ST100_Modify_e.proceedOperation_1: (*  *)
    IF xIN_NextStep AND (GetTick() - iStartProcessTimeMili) >= (iProcessTimeMili1) THEN
        iStartProcessTimeMili := GetTick();
        iOUT_Step             := ST100_Modify_e.proceedOperation_2;
		_bBewegung := FALSE;
		
    ELSIF __ISVALIDREF(Mover) THEN
        IF Mover.MoverAxis.isInPos THEN
            IF _bBewegung THEN
               // Mover.MoverAxis.RelMoveTo(_bBewegungDist);
            ELSE
                //Mover.MoverAxis.RelMoveTo(-_bBewegungDist);
            END_IF

            _bBewegung := NOT _bBewegung;
        END_IF;
    END_IF;

ST100_Modify_e.proceedOperation_2: (*  *)
    IF xIN_NextStep AND (GetTick() - iStartProcessTimeMili) >= (iProcessTimeMili2) THEN
        iOUT_Step := ST100_Modify_e.SYNC_MOVER_LEAVE;
    END_IF;

ST100_Modify_e.SYNC_MOVER_LEAVE:
    // The mover needs to be taken by MoverMan
    IF NOT __ISVALIDREF(Mover) THEN
        iOUT_Step := ST100_Unload_e.DONE;
    END_IF

(***** DONE *****)
ST100_Modify_e.DONE: (* Letzter Schritt  *)
    IF NOT xIN_AlarmAktiv THEN
        //AUTO
        IF (enIN_State = StateAUTO) AND xIN_RestartCYCL THEN
            iOUT_Step := ST100_Modify_e.START;
            //STEP / END / LEERFAHREN restart
        ELSIF (enIN_State < StateAUTO) AND (enIN_State >= enState.StateSTEP) AND xIN_RestartCYCL THEN
            iOUT_Step := ST100_Modify_e.START;
            //STEP / END / LEERFAHREN fertig
        ELSIF (enIN_State = StateREADY) THEN
            iOUT_Step := ST100_Modify_e.READY;
        END_IF;
    END_IF;

(************ ERROR *************)
ST100_Modify_e.ERROR: (* ERROR *) ;

END_CASE;

END_FUNCTION_BLOCK

// ---- POUs/20_AUTO/FileMan/FB_FileMan.TcPOU
FUNCTION_BLOCK FB_FileMan
VAR_INPUT
    sPathName   : STRING; //
    bSave       : BOOL;
    bLoad       : BOOL;
    sRefString  : POINTER TO STRING(2000);
    uiStringLen : DINT; // string length
END_VAR
VAR_OUTPUT
    bError   : BOOL;  // true when a FB is in error (all fb are mixed here)
    nErrorId : UDINT; // the error id from the fb in error (all fb are mixed here)

    currentState : INT; // current state of this FB, use it for debug
END_VAR
VAR
    fb_open  : FB_FileOpen;
    fb_write : FB_FileWrite;
    fb_read  : FB_FileRead;
    fb_close : FB_FileClose;
    hFile    : UINT; // file number holder for write operation
    state    : INT := 0;

    bOpState : INT;   //0 = saving operation, 1 = loading operation, other = error
    nMode    : DWORD; // file open monde, depending on the command

    byteRead : UDINT; //number of byte read so far
END_VAR


CASE state OF

0: (* wait for operation *)
    IF bSave THEN
        state    := 1;
        bOpState := 0;
        nMode    := FOPEN_MODEWRITE;
    ELSIF bLoad THEN
        state    := 1;
        bOpState := 1;
        nMode    := FOPEN_MODEREAD;
    END_IF

1: (* open *)
    fb_open(sNetId    := '',
            sPathName := sPathName,
            nMode     := nMode,
            ePath     := PATH_GENERIC,
            bExecute  := TRUE,
            tTimeout  := T#3S,
            bBusy     =>,
            bError    =>,
            nErrId    =>,
            hFile     => hFile);

    IF NOT fb_open.bBusy THEN
        fb_open(bExecute := FALSE);

        IF 0 = bOpState THEN
            state := 3;
        ELSIF 1 = bOpState THEN
            state    := 5;
            byteRead := 0;
        END_IF
    END_IF

3: (* write *)
    fb_write(sNetId     := '',
             hFile      := hFile,
             pWriteBuff := sRefString,
             cbWriteLen := TO_UDINT(uiStringLen),
             bExecute   := TRUE,
             tTimeout   := T#3S,
             bBusy      =>,
             bError     =>,
             nErrId     =>,
             cbWrite    =>);

    IF NOT fb_write.bBusy THEN
        fb_write(bExecute := FALSE);
        state := 10;
    END_IF

5: (* read 100 bytes *)
    IF fb_read.bEOF THEN
        state := 9;
    ELSE
        fb_read(sNetId    := '',
                hFile     := hFile,
                pReadBuff := sRefString,
                cbReadLen := TO_UDINT(uiStringLen),
                bExecute  := TRUE,
                tTimeout  :=,
                bBusy     =>,
                bError    =>,
                nErrId    =>,
                cbRead    => byteRead,
                bEOF      =>);

        state := 6;
    END_IF

6: (* open *)
    fb_read(bExecute := FALSE);
    state := 5;

9:
    state := 10;

10: (* open *)
    fb_close(sNetId   := '',
             hFile    := hFile,
             bExecute := TRUE,
             tTimeout := T#3S,
             bBusy    =>,
             bError   =>,
             nErrId   =>);

    IF NOT fb_close.bBusy AND NOT bSave AND NOT bLoad THEN
        fb_close(bExecute := FALSE);
        state := 0;
    END_IF

END_CASE

bError       := fb_open.bError OR fb_write.bError OR fb_read.bError OR fb_close.bError;
nErrorId     := fb_open.nErrId OR fb_write.nErrId OR fb_read.nErrId OR fb_close.nErrId;
currentState := state;

END_FUNCTION_BLOCK

// ---- POUs/20_AUTO/FileMan/FB_ReadJSON.TcPOU
{attribute 'c++_compatible'}
FUNCTION_BLOCK FB_ReadJSON IMPLEMENTS ITcJsonSaxHandler
VAR_INPUT
    myArrayInput1 : REFERENCE TO ARRAY[1..CONSt.STATION_NUMBER] OF DINT;
    myArrayInput2 : REFERENCE TO ARRAY[1..CONSt.STATION_NUMBER] OF DINT;
END_VAR
VAR_OUTPUT
END_VAR
VAR
    iArrayIndex : INT;
	iArrayNumber : INT := 0;
END_VAR

{attribute 'TcTypeSystem'}
{attribute 'no-analysis'}
{attribute 'c++_compatible'}
{attribute 'minimal_input_size' := '4'}
{attribute 'pack_mode' := '4'}
METHOD OnBool : HRESULT
VAR_INPUT
	value	: BOOL;
END_VAR
END_METHOD

{attribute 'TcTypeSystem'}
{attribute 'no-analysis'}
{attribute 'c++_compatible'}
{attribute 'minimal_input_size' := '4'}
{attribute 'pack_mode' := '4'}
METHOD OnDint : HRESULT
VAR_INPUT
	value	: DINT;
END_VAR
END_METHOD

{attribute 'TcTypeSystem'}
{attribute 'no-analysis'}
{attribute 'c++_compatible'}
{attribute 'minimal_input_size' := '4'}
{attribute 'pack_mode' := '4'}
METHOD OnEndArray : HRESULT
VAR_INPUT
	elementCount	: UDINT;
END_VAR
OnEndArray := S_OK;
END_METHOD

{attribute 'TcTypeSystem'}
{attribute 'no-analysis'}
{attribute 'c++_compatible'}
{attribute 'minimal_input_size' := '4'}
{attribute 'pack_mode' := '4'}
METHOD OnEndObject : HRESULT
VAR_INPUT
	memberCount	: UDINT;
END_VAR
OnEndObject := S_OK;
END_METHOD

{attribute 'TcTypeSystem'}
{attribute 'no-analysis'}
{attribute 'c++_compatible'}
{attribute 'minimal_input_size' := '4'}
{attribute 'pack_mode' := '4'}
METHOD OnKey : HRESULT
VAR_IN_OUT CONSTANT
	key	: STRING;
END_VAR
VAR_INPUT
	len	: UDINT;
END_VAR
OnKey := S_OK;
END_METHOD

{attribute 'TcTypeSystem'}
{attribute 'no-analysis'}
{attribute 'c++_compatible'}
{attribute 'minimal_input_size' := '4'}
{attribute 'pack_mode' := '4'}
METHOD OnLint : HRESULT
VAR_INPUT
	value	: LINT;
END_VAR
END_METHOD

{attribute 'TcTypeSystem'}
{attribute 'no-analysis'}
{attribute 'c++_compatible'}
{attribute 'minimal_input_size' := '4'}
{attribute 'pack_mode' := '4'}
METHOD OnLreal : HRESULT
VAR_INPUT
	value	: LREAL;
END_VAR
END_METHOD

{attribute 'TcTypeSystem'}
{attribute 'no-analysis'}
{attribute 'c++_compatible'}
{attribute 'minimal_input_size' := '4'}
{attribute 'pack_mode' := '4'}
METHOD OnNull : HRESULT
END_METHOD

{attribute 'TcTypeSystem'}
{attribute 'no-analysis'}
{attribute 'c++_compatible'}
{attribute 'minimal_input_size' := '4'}
{attribute 'pack_mode' := '4'}
METHOD OnRawNumber : HRESULT
VAR_IN_OUT CONSTANT
	value	: STRING;
END_VAR
VAR_INPUT
	len	: UDINT;
END_VAR
END_METHOD

{attribute 'TcTypeSystem'}
{attribute 'no-analysis'}
{attribute 'c++_compatible'}
{attribute 'minimal_input_size' := '4'}
{attribute 'pack_mode' := '4'}
METHOD OnStartArray : HRESULT
THIS^.iArrayIndex := 1;
THIS^.iArrayNumber := THIS^.iArrayNumber + 1;
OnStartArray := S_OK;
END_METHOD

{attribute 'TcTypeSystem'}
{attribute 'no-analysis'}
{attribute 'c++_compatible'}
{attribute 'minimal_input_size' := '4'}
{attribute 'pack_mode' := '4'}
METHOD OnStartObject : HRESULT
OnStartObject := S_OK;
END_METHOD

{attribute 'TcTypeSystem'}
{attribute 'no-analysis'}
{attribute 'c++_compatible'}
{attribute 'minimal_input_size' := '4'}
{attribute 'pack_mode' := '4'}
METHOD OnString : HRESULT
VAR_IN_OUT CONSTANT
	value	: STRING;
END_VAR
VAR_INPUT
	len	: UDINT;
END_VAR
END_METHOD

{attribute 'TcTypeSystem'}
{attribute 'no-analysis'}
{attribute 'c++_compatible'}
{attribute 'minimal_input_size' := '4'}
{attribute 'pack_mode' := '4'}
METHOD OnUdint : HRESULT
VAR_INPUT
	value	: UDINT;
END_VAR
IF THIS^.iArrayNumber = 1 THEN
    THIS^.myArrayInput1[THIS^.iArrayIndex] := TO_DINT(value);
    THIS^.iArrayIndex                      := THIS^.iArrayIndex + 1;
ELSIF THIS^.iArrayNumber = 2 THEN
    THIS^.myArrayInput2[THIS^.iArrayIndex] := TO_DINT(value);
    THIS^.iArrayIndex                      := THIS^.iArrayIndex + 1;
END_IF
OnUdint := S_OK;
END_METHOD

{attribute 'TcTypeSystem'}
{attribute 'no-analysis'}
{attribute 'c++_compatible'}
{attribute 'minimal_input_size' := '4'}
{attribute 'pack_mode' := '4'}
METHOD OnUlint : HRESULT
VAR_INPUT
	value	: ULINT;
END_VAR
END_METHOD

{attribute 'TcTypeSystem'}
{attribute 'no-analysis'}
{attribute 'c++_compatible'}
{attribute 'minimal_input_size' := '4'}
{attribute 'pack_mode' := '4'}
METHOD TcAddRef : UDINT
END_METHOD

{attribute 'TcTypeSystem'}
{attribute 'no-analysis'}
{attribute 'c++_compatible'}
{attribute 'minimal_input_size' := '4'}
{attribute 'pack_mode' := '4'}
METHOD TcQueryInterface : HRESULT
VAR_INPUT
	iid	: REFERENCE TO IID;
	pipItf	: POINTER TO PVOID;
END_VAR
END_METHOD

{attribute 'TcTypeSystem'}
{attribute 'no-analysis'}
{attribute 'c++_compatible'}
{attribute 'minimal_input_size' := '4'}
{attribute 'pack_mode' := '4'}
METHOD TcRelease : UDINT
END_METHOD

END_FUNCTION_BLOCK

// ---- POUs/20_AUTO/FileMan/LoadFromMemory.TcPOU
FUNCTION LoadFromMemory : BOOL
VAR_INPUT
    sData : REFERENCE TO STRING(2000);
END_VAR
VAR
    fbJson     : FB_JsonSaxReader;
    pJsonParse : FB_ReadJSON;

    i : int;
END_VAR

pJsonParse.myArrayInput1 REF= PERS.iStationTimeDef1;
pJsonParse.myArrayInput2 REF= PERS.iStationTimeDef2;
fbJson.Parse(sJson := sData, ipHdl := pJsonParse);

END_FUNCTION

// ---- POUs/20_AUTO/FileMan/SaveInMemory.TcPOU
FUNCTION SaveInMemory : BOOL
VAR_INPUT
    sData : REFERENCE TO STRING(2000);
END_VAR
VAR
    fbJson     : FB_JsonSaxWriter;
    i          : int;
END_VAR

fbJson.ResetDocument();
// global object
fbJson.StartObject();
fbJson.AddKey('StationTimeArray');

// array1
fbJson.StartObject();
fbJson.AddKey('StationTime1');
fbJson.StartArray();

FOR i := 1 TO CONST.STATION_NUMBER BY 1 DO
    fbJson.AddDint(PERS.iStationTimeDef1[i]);
END_FOR

fbJson.EndArray();

// array2
fbJson.AddKey('StationTime2');
fbJson.StartArray();

FOR i := 1 TO CONST.STATION_NUMBER BY 1 DO
    fbJson.AddDint(PERS.iStationTimeDef2[i]);
END_FOR

fbJson.EndArray();
fbJson.EndObject();

fbJson.EndObject();
// end global object

// end of file
sData := fbJson.GetDocument();

fbJson.ResetDocument();

END_FUNCTION

// ---- POUs/20_AUTO/Mover/FB_PieceHolder.TcPOU
FUNCTION_BLOCK FB_PieceHolder IMPLEMENTS IObject
VAR_INPUT
END_VAR
VAR_OUTPUT
END_VAR
VAR
	_lrPosOffset : LREAL; // current offset position
	
	_iID : INT := 0; // instance ID, is set during FB_Init using the value of _iInstanceCounter 
END_VAR
VAR_STAT
	_iInstanceCounter : INT := 1; // instance counter
END_VAR

METHOD Equals : BOOL
VAR_INPUT
    object : ANY;
END_VAR
Equals := THIS = object.pValue;
END_METHOD

METHOD FB_init : BOOL
VAR_INPUT
    bInitRetains : BOOL;  // if TRUE, the retain variables are initialized (warm start / cold start)
    bInCopyCode  : BOOL;  // if TRUE, the instance afterwards gets moved into the copy code (online change)
    offset       : LREAL; //position offset of the tool using this toolhead, a negative value represents a move on the left
END_VAR
THIS^._iID := THIS^._iInstanceCounter;
THIS^._iInstanceCounter := THIS^._iInstanceCounter +1;
THIS^.PosOffset := offset;
END_METHOD

PROPERTY PosOffset : LREAL
GET
PosOffset := _lrPosOffset;
END_GET
SET
_lrPosOffset := PosOffset;
END_SET
END_PROPERTY

METHOD ToString : STRING
VAR_INPUT
END_VAR
ToString := CONCAT('FB_PieceHolder_', TO_STRING(THIS^._iID));
END_METHOD

END_FUNCTION_BLOCK

// ---- POUs/20_AUTO/Mover/FB_SortMoverByPos.TcPOU
FUNCTION_BLOCK FB_SortMoverByPos EXTENDS FB_Sort
VAR_INPUT
END_VAR
VAR_OUTPUT
END_VAR
VAR
END_VAR

(* Please override this method so it returns:
* 0 : a == b
*-1 : a < b
* 1 : a > b
* which a and b are the ADDRESS of the 2 elements you want to compare
*)
METHOD Compare : DINT
VAR_INPUT
	a : PVOID;
	b : PVOID;
END_VAR
VAR
    MoverDict_a : MoverDict;
    MoverDict_b : MoverDict;
END_VAR
Tc2_System.MEMCPY(ADR(MoverDict_a), a, SIZEOF(MoverDict));
Tc2_System.MEMCPY(ADR(MoverDict_b), b, SIZEOF(MoverDict));

IF MoverDict_a.MoverPos < MoverDict_b.MoverPos THEN
    Compare := -1;

ELSIF MoverDict_a.MoverPos > MoverDict_b.MoverPos THEN
    Compare := 1;

ELSE
    Compare := 0;

END_IF
END_METHOD

END_FUNCTION_BLOCK

// ---- POUs/20_AUTO/ST100/FB_ABL_100.TcPOU
FUNCTION_BLOCK FB_ABL_100
(****************************************************************************************)
(*	TITEL				Bezeichnung Ablauf	    										*)
(*	Status				ungetestet                         								*)
(*  Version:			1.0																*)
(*	Beschrieb:			Ablaufbeschreibung												*)
(*																						*)
(*	Steps:																				*)
(*		RESET:=0		Reset der Station												*)
(* 		INIT:=100		Initialisieren													*)
(*		... 			...																*)
(*		READY:=999		Initialisiert, Bereit für Start									*)
(*		START:=1000		Start Zyklisch 													*)
(*		... 			...																*)
(*		DONE:=8000		Letzer Schritt													*)
(*		ERROR:=9000		ALARM/Fehler													*)
(* 	09.09.2019/Dj																		*)
(***********************************Revisionen*******************************************)
(*	dd.mm.yyyy   KZ    x.y			Beschrieb											*)
(****************************************************************************************)

VAR_INPUT
    xIN_Reset       : BOOL;          // Schrittkette zurücksetzen 
    xIN_Init        : BOOL;          // Initialisieren
    xIN_Quit        : BOOL;          // Fehler quittieren 
    xIN_Start       : BOOL;          // Startbefehl
    xIN_Sperre      : BOOL;          // FB Sperren 
    xIN_NextStep    : BOOL;          // Nächsten Schritt ausführen 
    xIN_AlarmAktiv  : BOOL;          // Anlage hat Alarm
    xIN_DryCycle    : BOOL;          // Fahren ohne Teile
    xIN_RestartCYCL : BOOL;          // Zyklus erneut starten im STEP, END, LEERFAHREN
    xIN_MoverInPos  : BOOL;          // Set this flag when a mover is in position and ready to be handled
    enIN_State      : enState;       // Status Anlage
    tIN_Timeout     : TIME := T#10s; // Timout

    pxFG_Freigabe : POINTER TO BOOL; //Freigabe von Station

    // Application specific
    iProcessTimeMili : UDINT := 5000; // user defined station duration, in milisecond
END_VAR
VAR_OUTPUT
    (* standart Ausgänge *)
    xOUT_ErrFlag   : BOOL;   // Error Flag 
    xOUT_Busy      : BOOL;   // Baustein befindet sich im Ablauf 
    xOUT_Done      : BOOL;   // Baustein hat den Ablauf beendet 		
    xOUT_Ready     : BOOL;   // Ready to begin, should be the same state as done	
    xOUT_Timeout   : BOOL;   // Timeout FB 
    xOUT_InitDone  : BOOL;   // initialisierung fertig
    xOUT_Wait      : BOOL;   // Wartet auf Bedingung
    xOUT_MoverFree : BOOL;   // The mover is free to move
    iOUT_Step      : INT;    // Aktueller Schritt 
    sOUT_Step      : STRING; // Aktueller Schritt but in string format
    bOUT_Error     : BYTE;   // Fehlernummer

    iOUT_ProcessCompletion : INT; //process completion, express in % (0-100)
END_VAR
VAR
    (* Standard *)
    (* Schritt *)
    iLastStep : INT; // Merker letzter Schritt 
    iPreStep  : INT; // Schritt zurück nach Alarm 
    iAktStep  : INT; // aktueller Schritt

    // Trigger Starten 
    rtSTART : R_TRIG;
    // Timer TimeOut 
    TON_Timeout : TON;

    (* Bausteine *)

    (* Spezial *)
    iStartProcessTimeMili : UDINT; // start of the processing time, accurate at 100ns 

END_VAR
VAR CONSTANT
END_VAR

(*******************************************************************)
(* Trigger  *)
(*******************************************************************)
(* Zurücksetzen *)
IF xIN_RESET THEN
    iPreStep  := ST100_e.RESET;
    iOUT_Step := ST100_e.RESET;
END_IF;

(* Error Quittieren *)
IF (bOUT_Error <> 0) AND xIN_Quit THEN
    xOUT_ErrFlag := FALSE;
    bOUT_Error   := 0;
    iOUT_Step    := iPreStep;
END_IF;

(*******************************************************************)
(* Timer *)
(*******************************************************************)
TON_Timeout(IN := xIN_NextStep AND (iLastStep = iOUT_Step) (*todo FG *) ,
            PT := tIN_Timeout);

(*******************************************************************)
(* Bausteine *)
(*******************************************************************)

(*******************************************************************)
(* OUTPUTS *)
(*******************************************************************)
// Error Flag 
xOUT_ErrFlag := (bOUT_Error <> 0);
// Baustein befindet sich im Ablauf 
xOUT_Busy := (iOUT_Step > ST100_e.READY) AND (iOUT_Step < ST100_e.DONE);
// Baustein hat den Ablauf beendet
xOUT_Done := (iOUT_Step = ST100_e.DONE);
// Process ready
xOUT_Ready := (iOUT_Step = ST100_e.READY);
// Timeout FB 				 		
xOUT_Timeout := TON_Timeout.Q;
// Itialisierung fertig			
xOUT_InitDone := (iOUT_Step = ST100_e.READY);
// Aktueller Schritt			
iOUT_Step := iOUT_Step; //Im Ablauf gesetzt		
sOUT_Step := TO_STRING(iOUT_Step);
//Fehlernummer	 
bOUT_Error := bOUT_Error; //Im Ablauf/FB gesetzt	
(* Warte (alle Schritte wo auf FG oder Teile gewartet wird) *)
xOUT_Wait := (iOUT_Step = ST100_e.DONE);

xOUT_MoverFree := iOUT_Step >= ST100_e.MOVER_FREE_OP AND iOUT_Step < ST100_e.MOVER_NEEDED_OP;

IF iAktStep < ST100_e.START THEN
    iOUT_ProcessCompletion := 0;
ELSIF iAktStep > ST100_e.DONE THEN
    iOUT_ProcessCompletion := getPercent(iPreStep, TO_INT(ST100_e.START), TO_INT(ST100_e.proceedOperation_2) + 1);
ELSIF ST100_e.DONE = iAktStep THEN
    iOUT_ProcessCompletion := 100;
ELSE
    // iOUT_ProcessCompletion := getPercent(iAktStep, TO_INT(ST100_e.START), TO_INT(ST100_e.releaseMover) + 1);
    IF iProcessTimeMili > 0 THEN
        IF iAktStep < ST100_e.proceedOperation_1 THEN
            iOUT_ProcessCompletion := 0;
        ELSIF iAktStep = ST100_e.proceedOperation_1 THEN
            iOUT_ProcessCompletion := TO_INT(((GetTick() - iStartProcessTimeMili) * 100) / iProcessTimeMili);
        ELSIF iAktStep = ST100_e.proceedOperation_2 THEN
            iOUT_ProcessCompletion := 50 + TO_INT(((GetTick() - iStartProcessTimeMili) * 100) / iProcessTimeMili);
        ELSE
            iOUT_ProcessCompletion := 50;
        END_IF
    ELSE
        iOUT_ProcessCompletion := 0;
    END_IF
END_IF

(*******************************************************************)
(* Ablauf *)
(*******************************************************************)

(* Sperren *)
IF xIN_Sperre THEN
    iPreStep  := ST100_e.RESET;
    iOUT_Step := ST100_e.RESET;
    RETURN;
END_IF;

(* Schritt Merker *)
IF iAktStep <> iOUT_Step THEN
    iLastStep := iAktStep;
    iAktStep  := iOUT_Step;
END_IF

(* START *)
rtSTART(CLK := xIN_Start);

(*******************************************************************)
(* Schrittkette  *)
(*******************************************************************)
CASE iOUT_Step OF

(***** RESET *****)
ST100_e.RESET: (* Schritt 0-99 *)
    //Initialisierungen
    //Start Init Ablauf
    IF xIN_Init THEN
        iOUT_Step := ST100_e.INIT;
        //Start Manu Ablauf
    ELSIF enIN_State = StateMANU AND xIN_NextStep THEN
        iOUT_Step := ST100_e.INIT;
    END_IF;

(***** INIT *****)
ST100_e.INIT: (* Grundstellung ? *)
    IF TRUE THEN
        iOUT_Step := ST100_e.READY;
    ELSE
        iOUT_Step := ST100_e.INIT;
    END_IF;

(***** READY / INIT DONE *****)
ST100_e.READY:        (* Start AUTO,END,LEER,STEP *)
    IF xIN_Start THEN //IF rtSTART.Q THEN
        iOUT_Step := ST100_e.START;
    END_IF

(***** START  ZYKLISCH *****)
ST100_e.START: (*  *)
    IF xIN_NextStep AND pxFG_Freigabe^ THEN
        iOUT_Step             := ST100_e.proceedOperation_1;
        iStartProcessTimeMili := GetTick();
    END_IF;

ST100_e.proceedOperation_1: (*  *)
    IF xIN_NextStep AND (GetTick() - iStartProcessTimeMili) >= (iProcessTimeMili / 2) THEN
        iOUT_Step := ST100_e.waitOnMover;
    END_IF;

ST100_e.waitOnMover: (*  *)
    IF xIN_NextStep AND xIN_MoverInPos THEN
        iStartProcessTimeMili := GetTick();
        iOUT_Step             := ST100_e.proceedOperation_2;
    END_IF;

ST100_e.proceedOperation_2: (*  *)
    IF xIN_NextStep AND (GetTick() - iStartProcessTimeMili) >= (iProcessTimeMili / 2) THEN
        iOUT_Step := ST100_e.DONE;
    END_IF;

(***** DONE *****)
ST100_e.DONE: (* Letzter Schritt  *)
    IF NOT xIN_AlarmAktiv THEN
        //AUTO
        IF (enIN_State = StateAUTO) AND xIN_RestartCYCL THEN
            iOUT_Step := ST100_e.START;
            //STEP / END / LEERFAHREN restart
        ELSIF (enIN_State < StateAUTO) AND (enIN_State >= enState.StateSTEP) AND xIN_RestartCYCL THEN
            iOUT_Step := ST100_e.START;
            //STEP / END / LEERFAHREN fertig
        ELSIF (enIN_State = StateREADY) THEN
            iOUT_Step := ST100_e.READY;
        END_IF;
    END_IF;

(************ ERROR *************)
ST100_e.ERROR: (* ERROR *) ;

END_CASE;

END_FUNCTION_BLOCK

// ---- POUs/20_AUTO/TOOL/EqualApproximately.TcPOU
(*approximatelyEqual gives whether the difference between a and b is smaller than the acceptable
 error (epsilon), determined by the larger of a or b. This means that the two values are 
"close enough", and we can say that they're approximately equal.*)
FUNCTION EqualApproximately
VAR_INPUT
    a       : LREAL;
    b       : LREAL;
    epsilon : LREAL;
END_VAR
VAR
END_VAR

IF ABS(a) < ABS(b) THEN
    EqualApproximately := ABS(a - b) <= (ABS(b) * epsilon);
ELSE
    EqualApproximately := ABS(a - b) <= (ABS(a) * epsilon);
END_IF

END_FUNCTION

// ---- POUs/20_AUTO/TOOL/EqualEssentially.TcPOU
(*essentiallyEqual gives whether the difference between a and b is smaller than the acceptable error (epsilon), 
determined by the smaller of a or b. This means that the values differ less than the acceptable difference in 
any calculation, so that perhaps they're not actually equal, but they're "essentially equal" (given the epsilon). *)
FUNCTION EqualEssentially : BOOL
VAR_INPUT
    a       : LREAL;
    b       : LREAL;
    epsilon : LREAL;
END_VAR
VAR
END_VAR

IF ABS(a) > ABS(b) THEN
    EqualEssentially := ABS(a - b) <= (ABS(b) * epsilon);
ELSE
    EqualEssentially := ABS(a - b) <= (ABS(a) * epsilon);
END_IF

END_FUNCTION

// ---- GlobalTextList.TcGTLO
TEXTLIST GlobalTextList
  373 = '%d'
  962 = '%f'
  999 = '%s'
  454 = '4'
  166 = 'Acceleration:'
  629 = 'AUTO'
  404 = 'Avg'
  101 = 'Current state'
  998 = 'Current state:'
  203 = 'END'
  557 = 'INIT'
  820 = 'LEER'
  905 = 'MANU'
  641 = 'Max'
  23 = 'Max speed:'
  386 = 'Min'
  590 = 'Mover 1 actual pos'
  716 = 'Mover 1 actual pos :'
  357 = 'Mover n°'
  310 = 'Mover n°%d'
  821 = 'Mover n°%s'
  679 = 'Navette 1 Pos'
  378 = 'PERS.iStationTimeDef[1]'
  375 = 'Piece holder:'
  639 = 'Process name:'
  964 = 'Process time :'
  566 = 'QUIT'
  849 = 'RESET TEMP COUNTER'
  832 = 'Save var'
  105 = 'SET'
  630 = 'Set all mover ApproachScenario'
  84 = 'Set all station time'
  137 = 'ST100'
  367 = 'ST105'
  965 = 'ST110'
  902 = 'ST115'
  633 = 'ST120'
  304 = 'ST125'
  610 = 'ST130'
  108 = 'ST135'
  328 = 'ST140'
  559 = 'ST145'
  406 = 'ST150'
  30 = 'ST155'
  326 = 'ST160'
  841 = 'ST165'
  619 = 'ST170'
  492 = 'ST175'
  422 = 'ST176'
  415 = 'ST180'
  710 = 'ST185'
  151 = 'ST190'
  960 = 'ST200'
  20 = 'ST210'
  526 = 'ST220'
  583 = 'ST230'
  75 = 'ST240'
  706 = 'ST250'
  364 = 'ST260'
  34 = 'ST270'
  69 = 'ST290'
  840 = 'ST300'
  729 = 'ST60'
  992 = 'ST70'
  939 = 'START'
  702 = 'Station name:'
  645 = 'STEP'
  457 = 'STOP'
  58 = 'Stop mover'
  242 = '[ms]'
END_TEXTLIST

// ---- VISUs/VISU_main.TcVIS
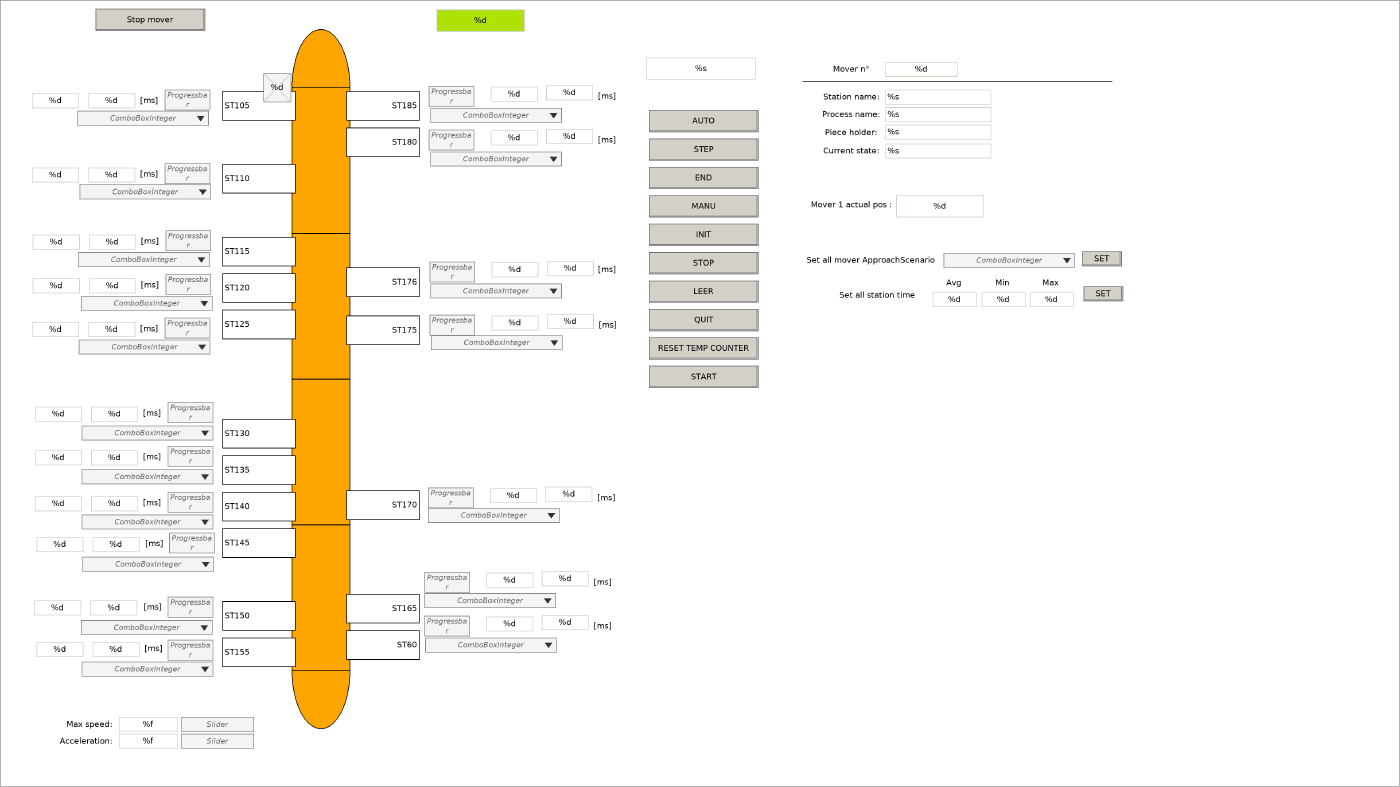
VISUALIZATION VISU_main  // 1920x1080
    Ellipse (400,840 80x160)
    Rectangle (400,720 80x200)
    Rectangle (400,520 80x200)
    Rectangle (400,320 80x200)
    Ellipse (400,40 80x160)
    Rectangle (400,120 80x200)
    Button (890,151 150x30), "AUTO", colour toggle: HMI.btArMain[0].on, input disabled if: HMI.btArMain[0].disable
        tap HMI.btArMain[0].button
    Button (890,190 150x30), "STEP", colour toggle: HMI.btArMain[1].on, input disabled if: HMI.btArMain[1].disable
        tap HMI.btArMain[1].button
    Button (890,229 150x30), "END", colour toggle: HMI.btArMain[2].on, input disabled if: HMI.btArMain[2].disable
        tap HMI.btArMain[2].button
    Button (890,307 150x30), "INIT", colour toggle: HMI.btArMain[4].on, input disabled if: HMI.btArMain[4].disable
        tap HMI.btArMain[4].button
    Button (890,346 150x30), "STOP", colour toggle: HMI.btArMain[5].disable, input disabled if: HMI.btArMain[5].disable
        tap HMI.btArMain[5].button
    Button (890,385 150x30), "LEER", colour toggle: HMI.btArMain[6].disable, input disabled if: HMI.btArMain[6].disable
        tap HMI.btArMain[6].button
    Button (890,424 150x30), "QUIT", colour toggle: HMI.btArMain[7].disable, input disabled if: HMI.btArMain[7].disable
        tap HMI.btArMain[7].button
    Button (890,463 150x30), "RESET TEMP COUNTER", colour toggle: HMI.btArMain[8].disable, input disabled if: HMI.btArMain[8].disable
        tap HMI.btArMain[8].button
    Button (890,268 150x30), "MANU", colour toggle: HMI.btArMain[3].on, input disabled if: HMI.btArMain[3].disable
        tap HMI.btArMain[3].button
    Textfield (886,79 150x30), "%s", text variable: _14_STATE.sStateDbg
    Button (890,502 150x30), "START", colour toggle: HMI.btArMain[9].disable, input disabled if: HMI.btArMain[9].disable
        tap HMI.btArMain[9].button
    Rectangle (475,175 100x40), "ST180", colour toggle: NOT PRG.st180_aut.xMoverPathFree
    Rectangle (475,367 100x40), "ST176", colour toggle: NOT PRG.st176_aut.xMoverPathFree
    Rectangle (475,433 100x40), "ST175", colour toggle: NOT PRG.st170_aut.xMoverPathFree
    Rectangle (475,673 100x40), "ST170", colour toggle: NOT PRG.st170_aut.xMoverPathFree
    Rectangle (475,815 100x40), "ST165", colour toggle: NOT PRG.st165_aut.xMoverPathFree
    Rectangle (475,865 100x40), "ST60", colour toggle: NOT PRG.st160_aut.xMoverPathFree
    Rectangle (305,875 100x40), "ST155", colour toggle: NOT PRG.st155_aut.xMoverPathFree
    Rectangle (475,125 100x40), "ST185", colour toggle: NOT PRG.st185_aut.xMoverPathFree
    Progressbar (588,178 62x28), variable: SIMU.iCompletionHMI[17]
    Progressbar (589,359 62x28), variable: SIMU.iCompletionHMI[16]
    Progressbar (589,432 62x28), variable: SIMU.iCompletionHMI[15]
    Progressbar (587,669 62x28), variable: SIMU.iCompletionHMI[14]
    Progressbar (582,785 62x28), variable: SIMU.iCompletionHMI[13]
    Progressbar (582,845 62x28), variable: SIMU.iCompletionHMI[12]
    Progressbar (230,878 62x28), variable: SIMU.iCompletionHMI[11]
    Progressbar (588,118 62x28), variable: SIMU.iCompletionHMI[18]
    Textfield (749,177 64x20), "%d", text variable: PERS.iStationTimeDef2[17]
        OnMouseDown: write the text variable via Default
    Label (805,177 55x30), "[ms]"
    Textfield (750,358 64x20), "%d", text variable: PERS.iStationTimeDef2[16]
        OnMouseDown: write the text variable via Default
    Label (805,355 55x30), "[ms]"
    Textfield (750,431 64x20), "%d", text variable: PERS.iStationTimeDef2[15]
        OnMouseDown: write the text variable via Default
    Label (806,431 55x30), "[ms]"
    Textfield (748,668 64x20), "%d", text variable: PERS.iStationTimeDef2[14]
        OnMouseDown: write the text variable via Default
    Label (804,668 55x30), "[ms]"
    Textfield (743,784 64x20), "%d", text variable: PERS.iStationTimeDef2[13]
        OnMouseDown: write the text variable via Default
    Label (799,784 55x30), "[ms]"
    Textfield (743,844 64x20), "%d", text variable: PERS.iStationTimeDef2[12]
        OnMouseDown: write the text variable via Default
    Label (799,844 55x30), "[ms]"
    Textfield (127,881 64x20), "%d", text variable: PERS.iStationTimeDef2[11]
        OnMouseDown: write the text variable via Default
    Label (183,875 55x30), "[ms]"
    Textfield (749,117 64x20), "%d", text variable: PERS.iStationTimeDef2[18]
        OnMouseDown: write the text variable via Default
    Label (805,117 55x30), "[ms]"
    Textfield (1229,268 120x30), "%d", text variable: MAIN.MoverMan._MoverList[1]._MoverAxis._CurrentPos
        OnMouseDown: write the text variable via Default
    Label (1080,266 146x30), "Mover 1 actual pos :"
    Textfield (599,13 120x30), "%d", text variable: PERS.iRecipeCurrent
        OnMouseDown: write the text variable via Default
    ComboBoxInteger (590,148 180x20), variable: MAIN.MoverMan._StationList[18]._ApproachScenario
    ComboBoxInteger (590,208 180x20), variable: MAIN.MoverMan._StationList[17]._ApproachScenario
    ComboBoxInteger (590,389 180x20), variable: MAIN.MoverMan._StationList[16]._ApproachScenario
    ComboBoxInteger (591,460 180x20), variable: MAIN.MoverMan._StationList[15]._ApproachScenario
    ComboBoxInteger (587,697 180x20), variable: MAIN.MoverMan._StationList[14]._ApproachScenario
    ComboBoxInteger (582,814 180x20), variable: MAIN.MoverMan._StationList[13]._ApproachScenario
    ComboBoxInteger (583,875 180x20), variable: MAIN.MoverMan._StationList[12]._ApproachScenario
    ComboBoxInteger (112,908 180x20), variable: MAIN.MoverMan._StationList[11]._ApproachScenario
    Rectangle (305,825 100x40), "ST150", colour toggle: NOT PRG.st150_aut.xMoverPathFree
    Progressbar (230,819 62x28), variable: SIMU.iCompletionHMI[10]
    Textfield (124,824 64x20), "%d", text variable: PERS.iStationTimeDef2[10]
        OnMouseDown: write the text variable via Default
    Label (182,818 55x30), "[ms]"
    ComboBoxInteger (111,851 180x20), variable: MAIN.MoverMan._StationList[10]._ApproachScenario
    Textfield (127,737 64x20), "%d", text variable: PERS.iStationTimeDef2[9]
        OnMouseDown: write the text variable via Default
    Label (184,731 55x30), "[ms]"
    Rectangle (305,725 100x40), "ST145", colour toggle: NOT PRG.st105_aut.xMoverPathFree
    Progressbar (232,731 62x28), variable: SIMU.iCompletionHMI[9]
    ComboBoxInteger (113,764 180x20), variable: MAIN.MoverMan._StationList[9]._ApproachScenario
    Textfield (125,681 64x20), "%d", text variable: PERS.iStationTimeDef2[8]
        OnMouseDown: write the text variable via Default
    Label (181,675 55x30), "[ms]"
    Rectangle (305,675 100x40), "ST140", colour toggle: NOT PRG.st140_aut.xMoverPathFree
    Progressbar (230,675 62x28), variable: SIMU.iCompletionHMI[8]
    ComboBoxInteger (112,706 180x20), variable: MAIN.MoverMan._StationList[8]._ApproachScenario
    Textfield (125,618 64x20), "%d", text variable: PERS.iStationTimeDef2[7]
        OnMouseDown: write the text variable via Default
    Label (181,612 55x30), "[ms]"
    Rectangle (305,625 100x40), "ST135", colour toggle: NOT PRG.st135_aut.xMoverPathFree
    Progressbar (230,612 62x28), variable: SIMU.iCompletionHMI[7]
    ComboBoxInteger (112,644 180x20), variable: MAIN.MoverMan._StationList[7]._ApproachScenario
    Textfield (125,558 64x20), "%d", text variable: PERS.iStationTimeDef2[6]
        OnMouseDown: write the text variable via Default
    Label (181,552 55x30), "[ms]"
    Rectangle (305,575 100x40), "ST130", colour toggle: NOT PRG.st130_aut.xMoverPathFree
    Progressbar (230,552 62x28), variable: SIMU.iCompletionHMI[6]
    ComboBoxInteger (112,584 180x20), variable: MAIN.MoverMan._StationList[6]._ApproachScenario
    Textfield (121,442 64x20), "%d", text variable: PERS.iStationTimeDef2[5]
        OnMouseDown: write the text variable via Default
    Label (177,436 55x30), "[ms]"
    Rectangle (305,425 100x40), "ST125", colour toggle: NOT PRG.st125_aut.xMoverPathFree
    Progressbar (226,436 62x28), variable: SIMU.iCompletionHMI[5]
    ComboBoxInteger (108,466 180x20), variable: MAIN.MoverMan._StationList[5]._ApproachScenario
    Textfield (122,382 64x20), "%d", text variable: PERS.iStationTimeDef2[4]
        OnMouseDown: write the text variable via Default
    Label (178,376 55x30), "[ms]"
    Rectangle (305,375 100x40), "ST120", colour toggle: NOT PRG.st120_aut.xMoverPathFree
    Progressbar (227,376 62x28), variable: SIMU.iCompletionHMI[4]
    ComboBoxInteger (111,406 180x20), variable: MAIN.MoverMan._StationList[4]._ApproachScenario
    Textfield (122,322 64x20), "%d", text variable: PERS.iStationTimeDef2[3]
        OnMouseDown: write the text variable via Default
    Label (178,316 55x30), "[ms]"
    Rectangle (305,325 100x40), "ST115", colour toggle: NOT PRG.st115_aut.xMoverPathFree
    Progressbar (227,316 62x28), variable: SIMU.iCompletionHMI[3]
    ComboBoxInteger (107,346 180x20), variable: MAIN.MoverMan._StationList[3]._ApproachScenario
    Textfield (121,230 64x20), "%d", text variable: PERS.iStationTimeDef2[2]
        OnMouseDown: write the text variable via Default
    Label (177,224 55x30), "[ms]"
    Rectangle (305,225 100x40), "ST110", colour toggle: NOT PRG.st110_aut.xMoverPathFree
    Progressbar (226,224 62x28), variable: SIMU.iCompletionHMI[2]
    ComboBoxInteger (109,253 180x20), variable: MAIN.MoverMan._StationList[2]._ApproachScenario
    Rectangle (305,125 100x40), "ST105", colour toggle: NOT PRG.st105_aut.xMoverPathFree
    Progressbar (226,123 62x28), variable: SIMU.iCompletionHMI[1]
    Textfield (121,128 64x20), "%d", text variable: PERS.iStationTimeDef2[1]
        OnMouseDown: write the text variable via Edit
    Label (177,123 55x30), "[ms]"
    ComboBoxInteger (106,152 180x20), variable: MAIN.MoverMan._StationList[1]._ApproachScenario
    ComboBoxInteger (1294,347 180x20), variable: MAIN.MoverMan.HMI_Scenario
    Label (1098,342 187x30), "Set all mover ApproachScenario"
    Button (1484,345 54x20), "SET"
        OnMouseDown: execute { MAIN.MoverMan.SetAllScenario(); }
    Label (1132,390 126x30), "Set all station time"
    Textfield (1279,401 60x20), "%d", text variable: MAIN.MoverMan.HMI_TimeAvg
        OnMouseDown: write the text variable via Default
    Label (1280,377 56x22), "Avg"
    Textfield (1346,401 60x20), "%d", text variable: MAIN.MoverMan.HMI_TimeMin
        OnMouseDown: write the text variable via Default
    Label (1347,377 56x22), "Min"
    Textfield (1412,401 60x20), "%d", text variable: MAIN.MoverMan.HMI_TimeMax
        OnMouseDown: write the text variable via Default
    Label (1413,377 56x22), "Max"
    Button (1486,393 54x20), "SET"
        OnMouseDown: execute { MAIN.MoverMan.SetAllTimers(ADR(PERS.iStationTimeDef1), 0); MAIN.MoverMan.SetAllTimers(ADR(PERS.iStationTimeDef2), 500); }
    Button (131,12 150x30), "Stop mover", colour toggle: MAIN.MoverMan.HMI_xStopMover
        toggle MAIN.MoverMan.HMI_xStopMover
    Label (1118,80 99x30), "Mover n°"
    Line (1101,111) (1525,111)
    Label (1118,118 99x30), "Station name:"
    Label (1118,142 99x30), "Process name:"
    Label (1118,167 99x30), "Piece holder:"
    Label (1118,192 99x30), "Current state:"
    Textfield (1214,85 99x20), "%d", text variable: MAIN.MoverMan.HMI_iSelMover
        OnMouseDown: write the text variable via Default
    Textfield (1214,123 145x20), "%s", text variable: MAIN.MoverMan._MoverList[MAIN.MoverMan.HMI_iSelMover].Station.ToString()
    Textfield (1214,147 145x20), "%s", text variable: MAIN.MoverMan._MoverList[MAIN.MoverMan.HMI_iSelMover].Station.Process.ToString()
    Textfield (1214,171 145x20), "%s"
    Textfield (1214,197 145x20), "%s", text variable: TO_STRING(MAIN.MoverMan._MoverList[MAIN.MoverMan.HMI_iSelMover]._State)
    Image (361,100 38x40), "%d", text variable: MAIN.MoverMan._MoverList[1]._ID, colour toggle: MAIN.MoverMan._SimuMoverList[1]._xStuck, invisible if: MAIN.MoverMan._MoverList[1]._MoverAxis._iID>CONST.MOVER_NUMBER, image: Custom.MoverSimu_final
        p3560616238: MAIN.MoverMan._MoverList[1]._MoverAxis.outSimuCurrentPos.x
        p2738717112: MAIN.MoverMan._MoverList[1]._MoverAxis.outSimuCurrentPos.y
        p2858320360: -MAIN.MoverMan._MoverList[1]._MoverAxis.outSimuCurrentRot
    Image (361,100 38x40), "%d", text variable: MAIN.MoverMan._MoverList[2]._ID, colour toggle: MAIN.MoverMan._SimuMoverList[2]._xStuck, invisible if: MAIN.MoverMan._MoverList[2]._MoverAxis._iID>CONST.MOVER_NUMBER, image: Custom.MoverSimu_final
        p3560616238: MAIN.MoverMan._MoverList[2]._MoverAxis.outSimuCurrentPos.x
        p2738717112: MAIN.MoverMan._MoverList[2]._MoverAxis.outSimuCurrentPos.y
        p2858320360: -MAIN.MoverMan._MoverList[2]._MoverAxis.outSimuCurrentRot
    Image (361,100 38x40), "%d", text variable: MAIN.MoverMan._MoverList[3]._ID, colour toggle: MAIN.MoverMan._SimuMoverList[3]._xStuck, invisible if: MAIN.MoverMan._MoverList[3]._MoverAxis._iID>CONST.MOVER_NUMBER, image: Custom.MoverSimu_final
        p3560616238: MAIN.MoverMan._MoverList[3]._MoverAxis.outSimuCurrentPos.x
        p2738717112: MAIN.MoverMan._MoverList[3]._MoverAxis.outSimuCurrentPos.y
        p2858320360: -MAIN.MoverMan._MoverList[3]._MoverAxis.outSimuCurrentRot
    Image (361,100 38x40), "%d", text variable: MAIN.MoverMan._MoverList[4]._ID, colour toggle: MAIN.MoverMan._SimuMoverList[4]._xStuck, invisible if: MAIN.MoverMan._MoverList[4]._MoverAxis._iID>CONST.MOVER_NUMBER, image: Custom.MoverSimu_final
        p3560616238: MAIN.MoverMan._MoverList[4]._MoverAxis.outSimuCurrentPos.x
        p2738717112: MAIN.MoverMan._MoverList[4]._MoverAxis.outSimuCurrentPos.y
        p2858320360: -MAIN.MoverMan._MoverList[4]._MoverAxis.outSimuCurrentRot
    Image (361,100 38x40), "%d", text variable: MAIN.MoverMan._MoverList[5]._ID, colour toggle: MAIN.MoverMan._SimuMoverList[5]._xStuck, invisible if: MAIN.MoverMan._MoverList[5]._MoverAxis._iID>CONST.MOVER_NUMBER, image: Custom.MoverSimu_final
        p3560616238: MAIN.MoverMan._MoverList[5]._MoverAxis.outSimuCurrentPos.x
        p2738717112: MAIN.MoverMan._MoverList[5]._MoverAxis.outSimuCurrentPos.y
        p2858320360: -MAIN.MoverMan._MoverList[5]._MoverAxis.outSimuCurrentRot
    Image (361,100 38x40), "%d", text variable: MAIN.MoverMan._MoverList[6]._ID, colour toggle: MAIN.MoverMan._SimuMoverList[6]._xStuck, invisible if: MAIN.MoverMan._MoverList[6]._MoverAxis._iID>CONST.MOVER_NUMBER, image: Custom.MoverSimu_final
        p3560616238: MAIN.MoverMan._MoverList[6]._MoverAxis.outSimuCurrentPos.x
        p2738717112: MAIN.MoverMan._MoverList[6]._MoverAxis.outSimuCurrentPos.y
        p2858320360: -MAIN.MoverMan._MoverList[6]._MoverAxis.outSimuCurrentRot
    Image (361,100 38x40), "%d", text variable: MAIN.MoverMan._MoverList[7]._ID, colour toggle: MAIN.MoverMan._SimuMoverList[7]._xStuck, invisible if: MAIN.MoverMan._MoverList[7]._MoverAxis._iID>CONST.MOVER_NUMBER, image: Custom.MoverSimu_final
        p3560616238: MAIN.MoverMan._MoverList[7]._MoverAxis.outSimuCurrentPos.x
        p2738717112: MAIN.MoverMan._MoverList[7]._MoverAxis.outSimuCurrentPos.y
        p2858320360: -MAIN.MoverMan._MoverList[7]._MoverAxis.outSimuCurrentRot
    Image (361,100 38x40), "%d", text variable: MAIN.MoverMan._MoverList[8]._ID, colour toggle: MAIN.MoverMan._SimuMoverList[8]._xStuck, invisible if: MAIN.MoverMan._MoverList[8]._MoverAxis._iID>CONST.MOVER_NUMBER, image: Custom.MoverSimu_final
        p3560616238: MAIN.MoverMan._MoverList[8]._MoverAxis.outSimuCurrentPos.x
        p2738717112: MAIN.MoverMan._MoverList[8]._MoverAxis.outSimuCurrentPos.y
        p2858320360: -MAIN.MoverMan._MoverList[8]._MoverAxis.outSimuCurrentRot
    Image (361,100 38x40), "%d", text variable: MAIN.MoverMan._MoverList[9]._ID, colour toggle: MAIN.MoverMan._SimuMoverList[9]._xStuck, invisible if: MAIN.MoverMan._MoverList[9]._MoverAxis._iID>CONST.MOVER_NUMBER, image: Custom.MoverSimu_final
        p3560616238: MAIN.MoverMan._MoverList[9]._MoverAxis.outSimuCurrentPos.x
        p2738717112: MAIN.MoverMan._MoverList[9]._MoverAxis.outSimuCurrentPos.y
        p2858320360: -MAIN.MoverMan._MoverList[9]._MoverAxis.outSimuCurrentRot
    Image (361,100 38x40), "%d", text variable: MAIN.MoverMan._MoverList[10]._ID, colour toggle: MAIN.MoverMan._SimuMoverList[10]._xStuck, invisible if: MAIN.MoverMan._MoverList[10]._MoverAxis._iID>CONST.MOVER_NUMBER, image: Custom.MoverSimu_final
        p3560616238: MAIN.MoverMan._MoverList[10]._MoverAxis.outSimuCurrentPos.x
        p2738717112: MAIN.MoverMan._MoverList[10]._MoverAxis.outSimuCurrentPos.y
        p2858320360: -MAIN.MoverMan._MoverList[10]._MoverAxis.outSimuCurrentRot
    Image (361,100 38x40), "%d", text variable: MAIN.MoverMan._MoverList[11]._ID, colour toggle: MAIN.MoverMan._SimuMoverList[11]._xStuck, invisible if: MAIN.MoverMan._MoverList[11]._MoverAxis._iID>CONST.MOVER_NUMBER, image: Custom.MoverSimu_final
        p3560616238: MAIN.MoverMan._MoverList[11]._MoverAxis.outSimuCurrentPos.x
        p2738717112: MAIN.MoverMan._MoverList[11]._MoverAxis.outSimuCurrentPos.y
        p2858320360: -MAIN.MoverMan._MoverList[11]._MoverAxis.outSimuCurrentRot
    Image (361,100 38x40), "%d", text variable: MAIN.MoverMan._MoverList[12]._ID, colour toggle: MAIN.MoverMan._SimuMoverList[12]._xStuck, invisible if: MAIN.MoverMan._MoverList[12]._MoverAxis._iID>CONST.MOVER_NUMBER, image: Custom.MoverSimu_final
        p3560616238: MAIN.MoverMan._MoverList[12]._MoverAxis.outSimuCurrentPos.x
        p2738717112: MAIN.MoverMan._MoverList[12]._MoverAxis.outSimuCurrentPos.y
        p2858320360: -MAIN.MoverMan._MoverList[12]._MoverAxis.outSimuCurrentRot
    Image (361,100 38x40), "%d", text variable: MAIN.MoverMan._MoverList[13]._ID, colour toggle: MAIN.MoverMan._SimuMoverList[13]._xStuck, invisible if: MAIN.MoverMan._MoverList[13]._MoverAxis._iID>CONST.MOVER_NUMBER, image: Custom.MoverSimu_final
        p3560616238: MAIN.MoverMan._MoverList[13]._MoverAxis.outSimuCurrentPos.x
        p2738717112: MAIN.MoverMan._MoverList[13]._MoverAxis.outSimuCurrentPos.y
        p2858320360: -MAIN.MoverMan._MoverList[13]._MoverAxis.outSimuCurrentRot
    Image (361,100 38x40), "%d", text variable: MAIN.MoverMan._MoverList[14]._ID, colour toggle: MAIN.MoverMan._SimuMoverList[14]._xStuck, invisible if: MAIN.MoverMan._MoverList[14]._MoverAxis._iID>CONST.MOVER_NUMBER, image: Custom.MoverSimu_final
        p3560616238: MAIN.MoverMan._MoverList[14]._MoverAxis.outSimuCurrentPos.x
        p2738717112: MAIN.MoverMan._MoverList[14]._MoverAxis.outSimuCurrentPos.y
        p2858320360: -MAIN.MoverMan._MoverList[14]._MoverAxis.outSimuCurrentRot
    Image (361,100 38x40), "%d", text variable: MAIN.MoverMan._MoverList[15]._ID, colour toggle: MAIN.MoverMan._SimuMoverList[15]._xStuck, invisible if: MAIN.MoverMan._MoverList[15]._MoverAxis._iID>CONST.MOVER_NUMBER, image: Custom.MoverSimu_final
        p3560616238: MAIN.MoverMan._MoverList[15]._MoverAxis.outSimuCurrentPos.x
        p2738717112: MAIN.MoverMan._MoverList[15]._MoverAxis.outSimuCurrentPos.y
        p2858320360: -MAIN.MoverMan._MoverList[15]._MoverAxis.outSimuCurrentRot
    Image (361,100 38x40), "%d", text variable: MAIN.MoverMan._MoverList[16]._ID, colour toggle: MAIN.MoverMan._SimuMoverList[16]._xStuck, invisible if: MAIN.MoverMan._MoverList[16]._MoverAxis._iID>CONST.MOVER_NUMBER, image: Custom.MoverSimu_final
        p3560616238: MAIN.MoverMan._MoverList[16]._MoverAxis.outSimuCurrentPos.x
        p2738717112: MAIN.MoverMan._MoverList[16]._MoverAxis.outSimuCurrentPos.y
        p2858320360: -MAIN.MoverMan._MoverList[16]._MoverAxis.outSimuCurrentRot
    Image (361,100 38x40), "%d", text variable: MAIN.MoverMan._MoverList[17]._ID, colour toggle: MAIN.MoverMan._SimuMoverList[17]._xStuck, invisible if: MAIN.MoverMan._MoverList[17]._MoverAxis._iID>CONST.MOVER_NUMBER, image: Custom.MoverSimu_final
        p3560616238: MAIN.MoverMan._MoverList[17]._MoverAxis.outSimuCurrentPos.x
        p2738717112: MAIN.MoverMan._MoverList[17]._MoverAxis.outSimuCurrentPos.y
        p2858320360: -MAIN.MoverMan._MoverList[17]._MoverAxis.outSimuCurrentRot
    Image (361,100 38x40), "%d", text variable: MAIN.MoverMan._MoverList[18]._ID, colour toggle: MAIN.MoverMan._SimuMoverList[18]._xStuck, invisible if: MAIN.MoverMan._MoverList[18]._MoverAxis._iID>CONST.MOVER_NUMBER, image: Custom.MoverSimu_final
        p3560616238: MAIN.MoverMan._MoverList[18]._MoverAxis.outSimuCurrentPos.x
        p2738717112: MAIN.MoverMan._MoverList[18]._MoverAxis.outSimuCurrentPos.y
        p2858320360: -MAIN.MoverMan._MoverList[18]._MoverAxis.outSimuCurrentRot
    Image (361,100 38x40), "%d", text variable: MAIN.MoverMan._MoverList[19]._ID, colour toggle: MAIN.MoverMan._SimuMoverList[19]._xStuck, invisible if: MAIN.MoverMan._MoverList[19]._MoverAxis._iID>CONST.MOVER_NUMBER, image: Custom.MoverSimu_final
        p3560616238: MAIN.MoverMan._MoverList[19]._MoverAxis.outSimuCurrentPos.x
        p2738717112: MAIN.MoverMan._MoverList[19]._MoverAxis.outSimuCurrentPos.y
        p2858320360: -MAIN.MoverMan._MoverList[19]._MoverAxis.outSimuCurrentRot
    Textfield (163,984 80x20), "%f", text variable: SIMU.lrSpeedMover
    Textfield (163,1007 80x20), "%f", text variable: SIMU.lrAccelMover
    Label (57,984 100x20), "Max speed:"
    Label (57,1007 100x20), "Acceleration:"
    Slider (248,984 100x20), variable: SIMU.lrSpeedMover, scale 1..50
    Slider (248,1007 100x20), variable: SIMU.lrAccelMoverSlider, scale 0.1..1
    Textfield (50,881 64x20), "%d", text variable: PERS.iStationTimeDef1[11]
        OnMouseDown: write the text variable via Default
    Textfield (47,824 64x20), "%d", text variable: PERS.iStationTimeDef1[10]
        OnMouseDown: write the text variable via Default
    Textfield (50,737 64x20), "%d", text variable: PERS.iStationTimeDef1[9]
        OnMouseDown: write the text variable via Default
    Textfield (48,681 64x20), "%d", text variable: PERS.iStationTimeDef1[8]
        OnMouseDown: write the text variable via Default
    Textfield (48,618 64x20), "%d", text variable: PERS.iStationTimeDef1[7]
        OnMouseDown: write the text variable via Default
    Textfield (48,558 64x20), "%d", text variable: PERS.iStationTimeDef1[6]
        OnMouseDown: write the text variable via Default
    Textfield (44,442 64x20), "%d", text variable: PERS.iStationTimeDef1[5]
        OnMouseDown: write the text variable via Default
    Textfield (45,382 64x20), "%d", text variable: PERS.iStationTimeDef1[4]
        OnMouseDown: write the text variable via Default
    Textfield (45,322 64x20), "%d", text variable: PERS.iStationTimeDef1[3]
        OnMouseDown: write the text variable via Default
    Textfield (44,230 64x20), "%d", text variable: PERS.iStationTimeDef1[2]
        OnMouseDown: write the text variable via Default
    Textfield (44,128 64x20), "%d", text variable: PERS.iStationTimeDef1[1]
        OnMouseDown: write the text variable via Edit
    Textfield (673,179 64x20), "%d", text variable: PERS.iStationTimeDef1[17]
        OnMouseDown: write the text variable via Default
    Textfield (674,360 64x20), "%d", text variable: PERS.iStationTimeDef1[16]
        OnMouseDown: write the text variable via Default
    Textfield (674,433 64x20), "%d", text variable: PERS.iStationTimeDef1[15]
        OnMouseDown: write the text variable via Default
    Textfield (672,670 64x20), "%d", text variable: PERS.iStationTimeDef1[14]
        OnMouseDown: write the text variable via Default
    Textfield (667,786 64x20), "%d", text variable: PERS.iStationTimeDef1[13]
        OnMouseDown: write the text variable via Default
    Textfield (667,846 64x20), "%d", text variable: PERS.iStationTimeDef1[12]
        OnMouseDown: write the text variable via Default
    Textfield (673,119 64x20), "%d", text variable: PERS.iStationTimeDef1[18]
        OnMouseDown: write the text variable via Default
END_VISUALIZATION
